FUNCTION_BLOCK TEST_CONGEN (* Test Internal Connection Generation: INT=>ANY, ANY=>ANY, ANY=>INT, INT=>INT *)
  (* Standard: 61499-2 *)
  (* Version 0.0, 2004-01-04, JHC, Rockwell Automation *)
  (* Compiler header: package fb.rt.test; import fb.rt.hmi.*; import fb.rt.math.*; *)
  (* Compiler Java IBM Jikes 1.06 *)
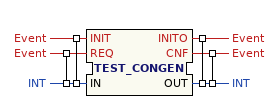
  EVENT_INPUT
    INIT WITH IN;
    REQ WITH IN;
  END_EVENT
  EVENT_OUTPUT
    INITO WITH OUT;
    CNF WITH OUT;
  END_EVENT
  VAR_INPUT
    IN : INT;
  END_VAR
  VAR_OUTPUT
    OUT : INT;
  END_VAR
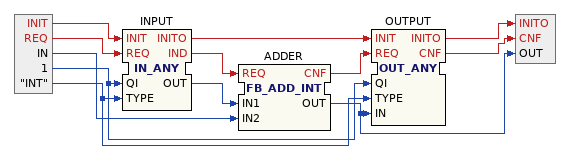
  FBS
    ADDER : FB_ADD_INT;
    INPUT : IN_ANY;
    OUTPUT : OUT_ANY;
  END_FBS
  EVENT_CONNECTIONS
    INIT TO INPUT.INIT;
    INPUT.INITO TO OUTPUT.INIT;
    OUTPUT.INITO TO INITO;
    REQ TO INPUT.REQ;
    OUTPUT.CNF TO CNF;
    INPUT.IND TO ADDER.REQ;
    ADDER.CNF TO OUTPUT.REQ;
  END_CONNECTIONS
  DATA_CONNECTIONS
    1 TO INPUT.QI;
    "INT" TO INPUT.TYPE;
    1 TO OUTPUT.QI;
    "INT" TO OUTPUT.TYPE;
    INPUT.OUT TO ADDER.IN1;
    IN TO ADDER.IN2;
    ADDER.OUT TO OUTPUT.IN;
    ADDER.OUT TO OUT;
  END_CONNECTIONS
END_FUNCTION_BLOCK
